// Mitsubishi GX Works2 project: PLC_Group15   PLC: FX3G

// global labels: Global1
VAR_GLOBAL
  StartworkingDay AT X010 : BOOL;
  insertOrange AT D8280 : REAL;
END_VAR
VAR_GLOBAL CONSTANT
  Muiltipy1 : WORD := 100;
  multiply1 : INT;
  divideBy2 : REAL := 2.0;
END_VAR
VAR_GLOBAL
  light AT Y010 : BOOL;
  SampleClemetine AT M2 : BOOL;
  sampleClementine AT D8281 : REAL;
END_VAR
VAR_GLOBAL CONSTANT
  multiply2 : REAL := 100.0;
END_VAR
VAR_GLOBAL
  clemetineInStoreAfterMultiply AT D4005 : REAL;
  checkProportion AT Y006 : BOOL;
  SamplePummels AT X004 : BOOL;
END_VAR
VAR_GLOBAL CONSTANT
  multiply3 : REAL := 100.0;
END_VAR
VAR_GLOBAL
  checkProportion2 AT M42 : BOOL;
  insertClementine AT D8281 : REAL;
  insertPummels AT D8281 : REAL;
  holding AT Y006 : BOOL;
  holding2 AT Y011 : BOOL;
  workingDayLight AT Y010 : BOOL;
  collectFruits AT X002 : BOOL;
END_VAR
VAR_GLOBAL CONSTANT
  washingTimer : REAL := 300.0;
END_VAR
VAR_GLOBAL
  lightOfWashing AT Y005 : BOOL;
  StartingWash AT M7 : BOOL;
END_VAR
VAR_GLOBAL CONSTANT
  const100 : REAL := 100.0;
END_VAR
VAR_GLOBAL
  BiggerThan100 AT M0 : BOOL;
  TakeOnly100 AT M0 : BOOL;
END_VAR
VAR_GLOBAL CONSTANT
  Take100 : REAL := 100.0;
  Take50 : REAL := 50.0;
END_VAR
VAR_GLOBAL
  TurningOnWash AT X002 : BOOL;
  SampleOrange AT M1 : BOOL;
  OrangeSample AT M1 : BOOL;
  ClementineSample AT M2 : BOOL;
  PummelSample AT M3 : BOOL;
  TurnigWashOn AT M4 : BOOL;
  Check100Oranges AT M5 : BOOL;
  Move100 AT M6 : BOOL;
  StartingWash2 AT M7 : BOOL;
  TurningLightWashOn AT M4 : BOOL;
  LessThan100 AT M0 : BOOL;
  MoveLessThan100 AT M8 : BOOL;
END_VAR
VAR_GLOBAL CONSTANT
  Add_150_to_washing_container : INT := 150;
END_VAR
VAR_GLOBAL
  MoveFromStorageToWashing AT X002 : BOOL;
  MoveFromWashingToPress AT X001 : BOOL;
  Collect_Fruits AT X001 : BOOL;
  Keep_Y1_ON AT M18 : BOOL;
  LightForCollecting AT Y001 : BOOL;
END_VAR
VAR_GLOBAL CONSTANT
  Add_100_Oranges : REAL := 100.0;
  Add_50_Clementines : REAL := 50.0;
  Add_50_Pummels : REAL := 50.0;
END_VAR
VAR_GLOBAL
  MoveFruitsToPressContainer AT M9 : BOOL;
  StartPressingProcess AT X011 : BOOL;
  CountingClicks AT CC1 : BOOL;
END_VAR
VAR_GLOBAL CONSTANT
  NumberOfClicks : REAL := 2.0;
END_VAR
VAR_GLOBAL
  Turn_Of_Y1 AT M18 : BOOL;
  StartQA AT X003 : BOOL;
  Sample_AnalogInput2 AT M10 : BOOL;
  CheckValueRange AT M11 : BOOL;
END_VAR
VAR_GLOBAL CONSTANT
  LowerBound : INT := 1;
END_VAR
VAR_GLOBAL
  GE_Than1 AT M12 : BOOL;
  CheckValueRange1 AT M11 : BOOL;
  CheckValueRange2 AT M13 : BOOL;
END_VAR
VAR_GLOBAL CONSTANT
  UpperBound : INT := 5;
  Const1 : REAL := 1.0;
  Const5 : REAL := 5.0;
END_VAR
VAR_GLOBAL
  LE_Than5 AT M14 : BOOL;
  If_M12_ON AT M12 : BOOL;
  If_M14_ON AT M14 : BOOL;
  Timer_Y4_Light AT TC1 : BOOL;
END_VAR
VAR_GLOBAL CONSTANT
  TimerValue : REAL := 500.0;
END_VAR
VAR_GLOBAL
  QA_Light AT Y004 : BOOL;
  Move_Juice_To_Storage AT M15 : BOOL;
  Greater_Than5 AT M12 : BOOL;
  Lower_Than1 AT M14 : BOOL;
  Didnt_Pass_QA AT M16 : BOOL;
  Pass_QA AT M16 : BOOL;
  SampleAgain AT M17 : BOOL;
  Shutting_Y1_Off AT M18 : BOOL;
  FlashingLightsOn AT M18 : BOOL;
  Y2Flash AT Y002 : BOOL;
  Y2Counter AT TC2 : BOOL;
  Turn_Off_Y2 AT TS2 : BOOL;
END_VAR
VAR_GLOBAL CONSTANT
  Const300 : INT := 300;
END_VAR
VAR_GLOBAL
  TurningLightsOn AT M19 : BOOL;
  Y3Counter AT TC3 : BOOL;
  Turn_Off_Y3 AT TS3 : BOOL;
  TurningLightsOff AT TS3 : BOOL;
  CheckValueRange3 AT M20 : BOOL;
  CheckValueRange4 AT M21 : BOOL;
  Greater_Than5_2 AT M22 : BOOL;
  Y3FlashON AT Y003 : BOOL;
  Lower_Than1_22 AT M23 : BOOL;
END_VAR
VAR_GLOBAL CONSTANT
  Const0 : REAL;
END_VAR
VAR_GLOBAL
  NoOrangesInStore AT M24 : BOOL;
  Loop AT M25 : BOOL;
  CheckIfOrange0 AT M26 : BOOL;
  TruncateWashingContainers AT M27 : BOOL;
  TruncateAllFruitStores AT M28 : BOOL;
  Truncate_All_Fruit_Stores AT M28 : BOOL;
  NoOrangesLeft AT M24 : BOOL;
  emergencyExit AT X007 : BOOL;
  X7_Light AT M29 : BOOL;
  MoveToJuiceContainer AT M30 : BOOL;
  EmptyJuice AT M31 : BOOL;
  StartTimerForStorage AT M32 : BOOL;
  CheckJuice AT M33 : BOOL;
  QA1 AT M34 : BOOL;
  Truncate_Juice_Container AT M35 : BOOL;
  insertOranges AT D3000 : REAL;
  OrangesInStore AT D3002 : REAL;
  halfOrange AT D1106 : REAL;
  insertPummel AT D5000 : REAL;
  insertClementines AT D4000 : REAL;
  ClemetinesWashingContainer AT D6002 : REAL;
  PummelsWashingContainer AT D6004 : REAL;
  OrangesWashingContainer AT D6000 : REAL;
  PressContainer AT D6010 : REAL;
  JuiceContainer AT D6012 : REAL;
  SampleAnalogInput2 AT D8281 : INT;
  SaveAnalogOutput AT D6014 : REAL;
  AnalogOutput AT D8282 : INT;
  OrangesAndClementines AT D6008 : REAL;
  StorageContainer AT D6016 : REAL;
  ClementinesInStore AT D4050 : REAL;
  pummelInStore AT D5050 : REAL;
END_VAR
VAR_GLOBAL CONSTANT
  Const2 : INT := 2;
END_VAR
VAR_GLOBAL
  countingWash AT TC0 : BOOL;
END_VAR
VAR_GLOBAL CONSTANT
  Const500 : INT := 500;
END_VAR
VAR_GLOBAL
  Y10_light AT TC4 : BOOL;
  end_day_light AT Y010 : BOOL;
END_VAR
VAR_GLOBAL CONSTANT
  Const_half : INT := 5;
END_VAR
VAR_GLOBAL
  M19Counter AT TC5 : BOOL;
  MoveToJuicer AT TS5 : BOOL;
  SecondQA AT M36 : BOOL;
  Didnt_Pass_QA2 AT M37 : BOOL;
  PassQA_Light AT M38 : BOOL;
  Turn_Lights_Off AT M39 : BOOL;
  Start_QA_Stage AT M40 : BOOL;
  checkProportion1 AT M41 : BOOL;
  checkProportionClementine AT M41 : BOOL;
  checkProportion_2 AT M42 : BOOL;
  Initialize_Y1 AT M43 : BOOL;
  Day_Started AT M44 : BOOL;
  Day_Ended AT M45 : BOOL;
  Initialize_Y10 AT M43 : BOOL;
  Check AT M50 : BOOL;
  MoveToPress AT M45 : BOOL;
  checkTiming AT M51 : BOOL;
  CountingClicksForX11 AT CS1 : BOOL;
  SecondQA_Counter AT CC2 : BOOL;
  CountingWash2 AT TS0 : BOOL;
  SecondQACounter AT CS2 : BOOL;
END_VAR
VAR_GLOBAL CONSTANT
  Const404 : REAL := 404.5;
  Const30 : INT := 30;
  Const10000 : REAL := 10000.0;
END_VAR
VAR_GLOBAL
  Y4Light AT TS1 : BOOL;
END_VAR
VAR_GLOBAL CONSTANT
  Const50 : INT := 50;
END_VAR
VAR_GLOBAL
  Mid_juice_truncate AT M52 : BOOL;
  Close_Y10 AT TS4 : BOOL;
  ClosingTime AT M55 : BOOL;
  FinishCheck1 AT M55 : BOOL;
  FinishCheck2 AT M56 : BOOL;
  MoveAndEmptyPress AT M57 : BOOL;
  FinishedSecondQA AT M58 : BOOL;
  FirstQADone AT M59 : BOOL;
  FirstQA2Done AT M60 : BOOL;
  SecondQADone AT M60 : BOOL;
  SecondQA2Done AT M61 : BOOL;
  tc9 AT TC9 : BOOL;
  ts9 AT TS9 : BOOL;
  Lamp6 AT Y006 : BOOL;
END_VAR
VAR_GLOBAL CONSTANT
  Const_6 : REAL := 6;
  Const_6_int : INT := 6;
  Const_100 : REAL := 100;
END_VAR
VAR_GLOBAL
  FillJuice AT X000 : BOOL;
  StartFillJuice AT M62 : BOOL;
END_VAR
VAR_GLOBAL CONSTANT
  Const_1_5 : REAL := 1.5;
END_VAR
VAR_GLOBAL
  TotalBottles AT D1108 : REAL;
  TimeToFillBottles AT D1110 : INT;
END_VAR
VAR_GLOBAL CONSTANT
  Const_10_int : INT := 10;
  Const_10 : REAL := 10;
END_VAR
VAR_GLOBAL
  checkLessThan10 AT M63 : BOOL;
  LessThan10 AT M64 : BOOL;
  StartLightFillBottles AT M65 : BOOL;
END_VAR
VAR_GLOBAL CONSTANT
  blinkTime : INT := 5;
END_VAR
VAR_GLOBAL
  resetBlink AT M66 : BOOL;
  blink1 AT M67 : BOOL;
  blink2 AT M68 : BOOL;
  tc6 AT TC6 : BOOL;
  ts6 AT TS6 : BOOL;
  tc7 AT TC7 : BOOL;
  ts7 AT TS7 : BOOL;
  tc8 AT TC8 : BOOL;
  ts8 AT TS8 : BOOL;
  Start2blinks AT M69 : BOOL;
  EQto0 AT M70 : BOOL;
END_VAR
VAR_GLOBAL CONSTANT
  Const400 : REAL := 400;
END_VAR

// task Task_01 (event TRUE, interval 0, priority 31): POU_01

PROGRAM POU_01
(* structured ladder/FBD written out as ST: instructions are called as NAME(EN, inputs, outputs); _pN, _eN, _tN stand for wires *)
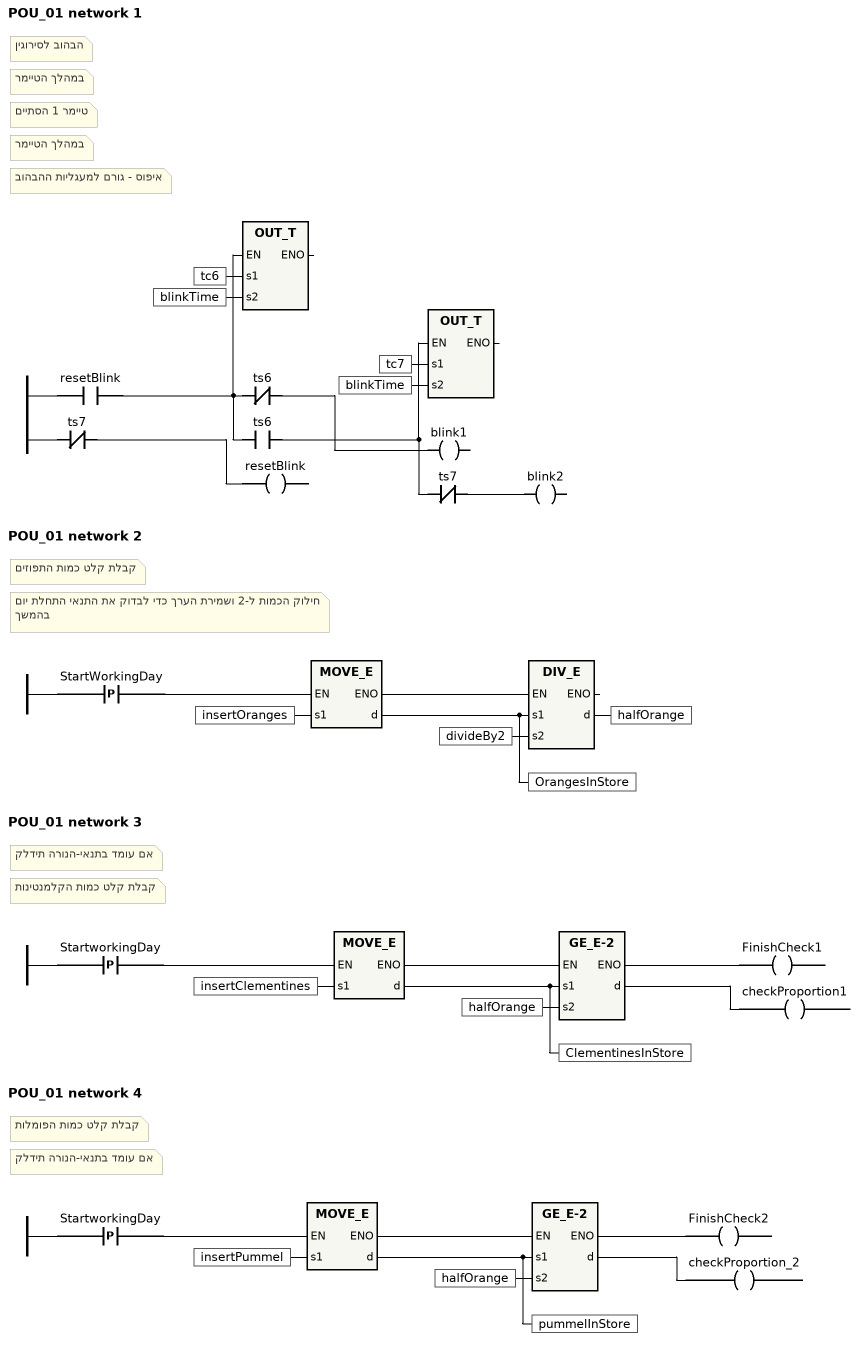
(* network 1 *)
(* הבהוב לסירוגין *)
(* במהלך הטיימר *)
(* טיימר 1 הסתיים *)
(* במהלך הטיימר *)
(* איפוס - גורם למעגליות ההבהוב *)
OUT_T(resetBlink, tc6, blinkTime);
blink1 := resetBlink AND NOT ts6;
_p1 := resetBlink AND ts6;
OUT_T(_p1, tc7, blinkTime);
blink2 := _p1 AND NOT ts7;
resetBlink := NOT ts7;
(* network 2 *)
(* קבלת קלט כמות התפוזים *)
(* חילוק הכמות ל-2 ושמירת הערך כדי לבדוק את התנאי התחלת יום בהמשך *)
_e1 := MOVE_E(LDP(TRUE, StartWorkingDay), insertOranges, OrangesInStore);
DIV_E(_e1, OrangesInStore, divideBy2, halfOrange);
(* network 3 *)
(* אם עומד בתנאי-הנורה תידלק *)
(* קבלת קלט כמות הקלמנטינות *)
_e1 := MOVE_E(LDP(TRUE, StartworkingDay), insertClementines, ClementinesInStore);
_e3 := GE_E(_e1, ClementinesInStore, halfOrange, _t2);
FinishCheck1 := _e3;
checkProportion1 := _t2;
(* network 4 *)
(* קבלת קלט כמות הפומלות *)
(* אם עומד בתנאי-הנורה תידלק *)
_e1 := MOVE_E(LDP(TRUE, StartworkingDay), insertPummel, pummelInStore);
_e3 := GE_E(_e1, pummelInStore, halfOrange, _t2);
FinishCheck2 := _e3;
checkProportion_2 := _t2;
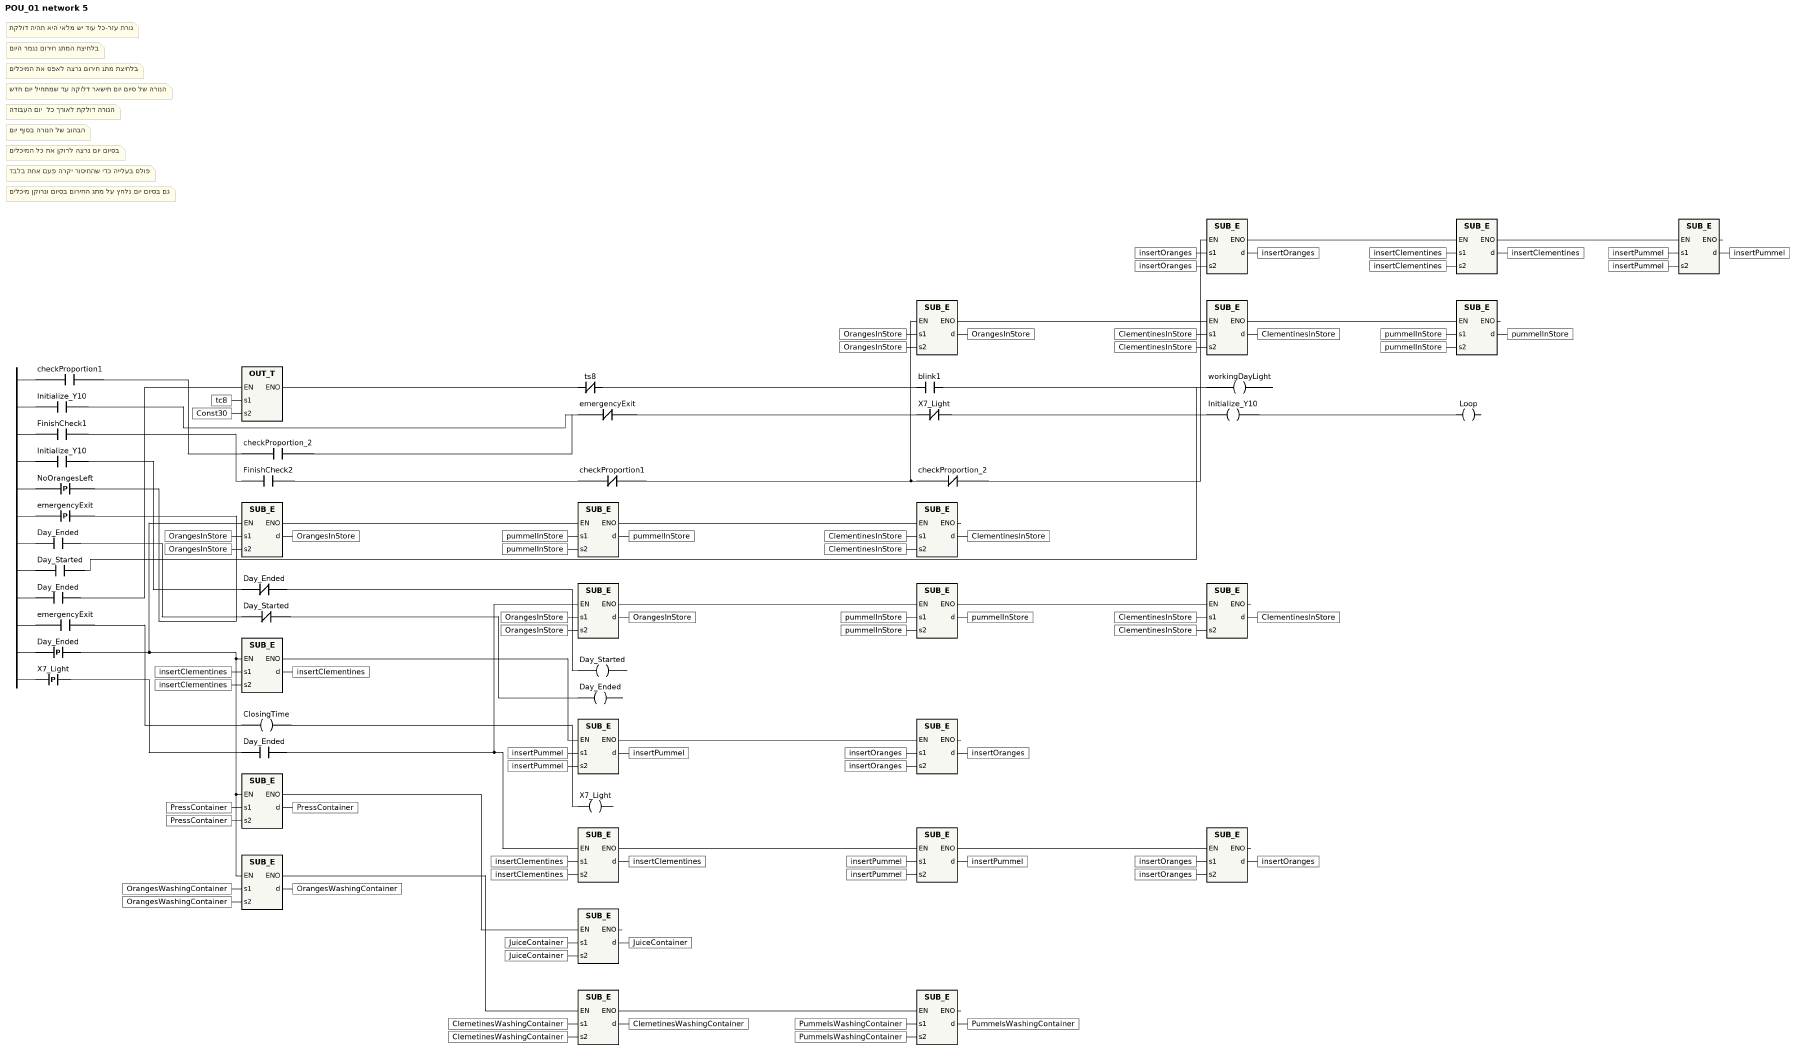
(* network 5 *)
(* נורת עזר-כל עוד יש מלאי היא תהיה דולקת *)
(* בלחיצת המתג חירום נגמר היום *)
(* בלחיצת מתג חירום נרצה לאפס את המיכלים *)
(* הנורה של סיום יום תישאר דלוקה עד שמתחיל יום חדש *)
(* הנורה דולקת לאורך כל  יום העבודה *)
(* הבהוב של הנורה בסוף יום *)
(* בסיום יום נרצה לרוקן את כל המיכלים *)
(* פולס בעלייה כדי שהחיסור יקרה פעם אחת בלבד *)
(* גם בסיום יום נלחץ על מתג החירום בסיום ונרוקן מיכלים *)
_p1 := (((checkProportion1 AND checkProportion_2) OR Initialize_Y10) AND NOT emergencyExit) AND NOT X7_Light;
Initialize_Y10 := _p1;
Loop := _p1;
_p2 := FinishCheck1 AND FinishCheck2 AND NOT checkProportion1;
_e3 := SUB_E(_p2 AND NOT checkProportion_2, insertOranges, insertOranges, insertOranges);
_e4 := SUB_E(_e3, insertClementines, insertClementines, insertClementines);
SUB_E(_e4, insertPummel, insertPummel, insertPummel);
_e5 := SUB_E(_p2, OrangesInStore, OrangesInStore, OrangesInStore);
_e6 := SUB_E(_e5, ClementinesInStore, ClementinesInStore, ClementinesInStore);
SUB_E(_e6, pummelInStore, pummelInStore, pummelInStore);
Day_Started := Initialize_Y10 AND NOT Day_Ended;
Day_Ended := (LDP(TRUE, NoOrangesLeft) OR LDP(TRUE, emergencyExit) OR Day_Ended) AND NOT Day_Started;
_e7 := OUT_T(Day_Ended, tc8, Const30);
workingDayLight := Day_Started OR (_e7 AND NOT ts8 AND blink1);
ClosingTime := emergencyExit;
X7_Light := emergencyExit;
_p8 := LDP(TRUE, Day_Ended);
_e9 := SUB_E(_p8, OrangesInStore, OrangesInStore, OrangesInStore);
_e10 := SUB_E(_e9, pummelInStore, pummelInStore, pummelInStore);
SUB_E(_e10, ClementinesInStore, ClementinesInStore, ClementinesInStore);
_e11 := SUB_E(_p8, insertClementines, insertClementines, insertClementines);
_e12 := SUB_E(_e11, insertPummel, insertPummel, insertPummel);
SUB_E(_e12, insertOranges, insertOranges, insertOranges);
_e13 := SUB_E(_p8, OrangesWashingContainer, OrangesWashingContainer, OrangesWashingContainer);
_e14 := SUB_E(_e13, ClemetinesWashingContainer, ClemetinesWashingContainer, ClemetinesWashingContainer);
SUB_E(_e14, PummelsWashingContainer, PummelsWashingContainer, PummelsWashingContainer);
_e15 := SUB_E(_p8, PressContainer, PressContainer, PressContainer);
SUB_E(_e15, JuiceContainer, JuiceContainer, JuiceContainer);
_p16 := LDP(TRUE, X7_Light) AND Day_Ended;
_e17 := SUB_E(_p16, OrangesInStore, OrangesInStore, OrangesInStore);
_e18 := SUB_E(_e17, pummelInStore, pummelInStore, pummelInStore);
SUB_E(_e18, ClementinesInStore, ClementinesInStore, ClementinesInStore);
_e19 := SUB_E(_p16, insertClementines, insertClementines, insertClementines);
_e20 := SUB_E(_e19, insertPummel, insertPummel, insertPummel);
SUB_E(_e20, insertOranges, insertOranges, insertOranges);
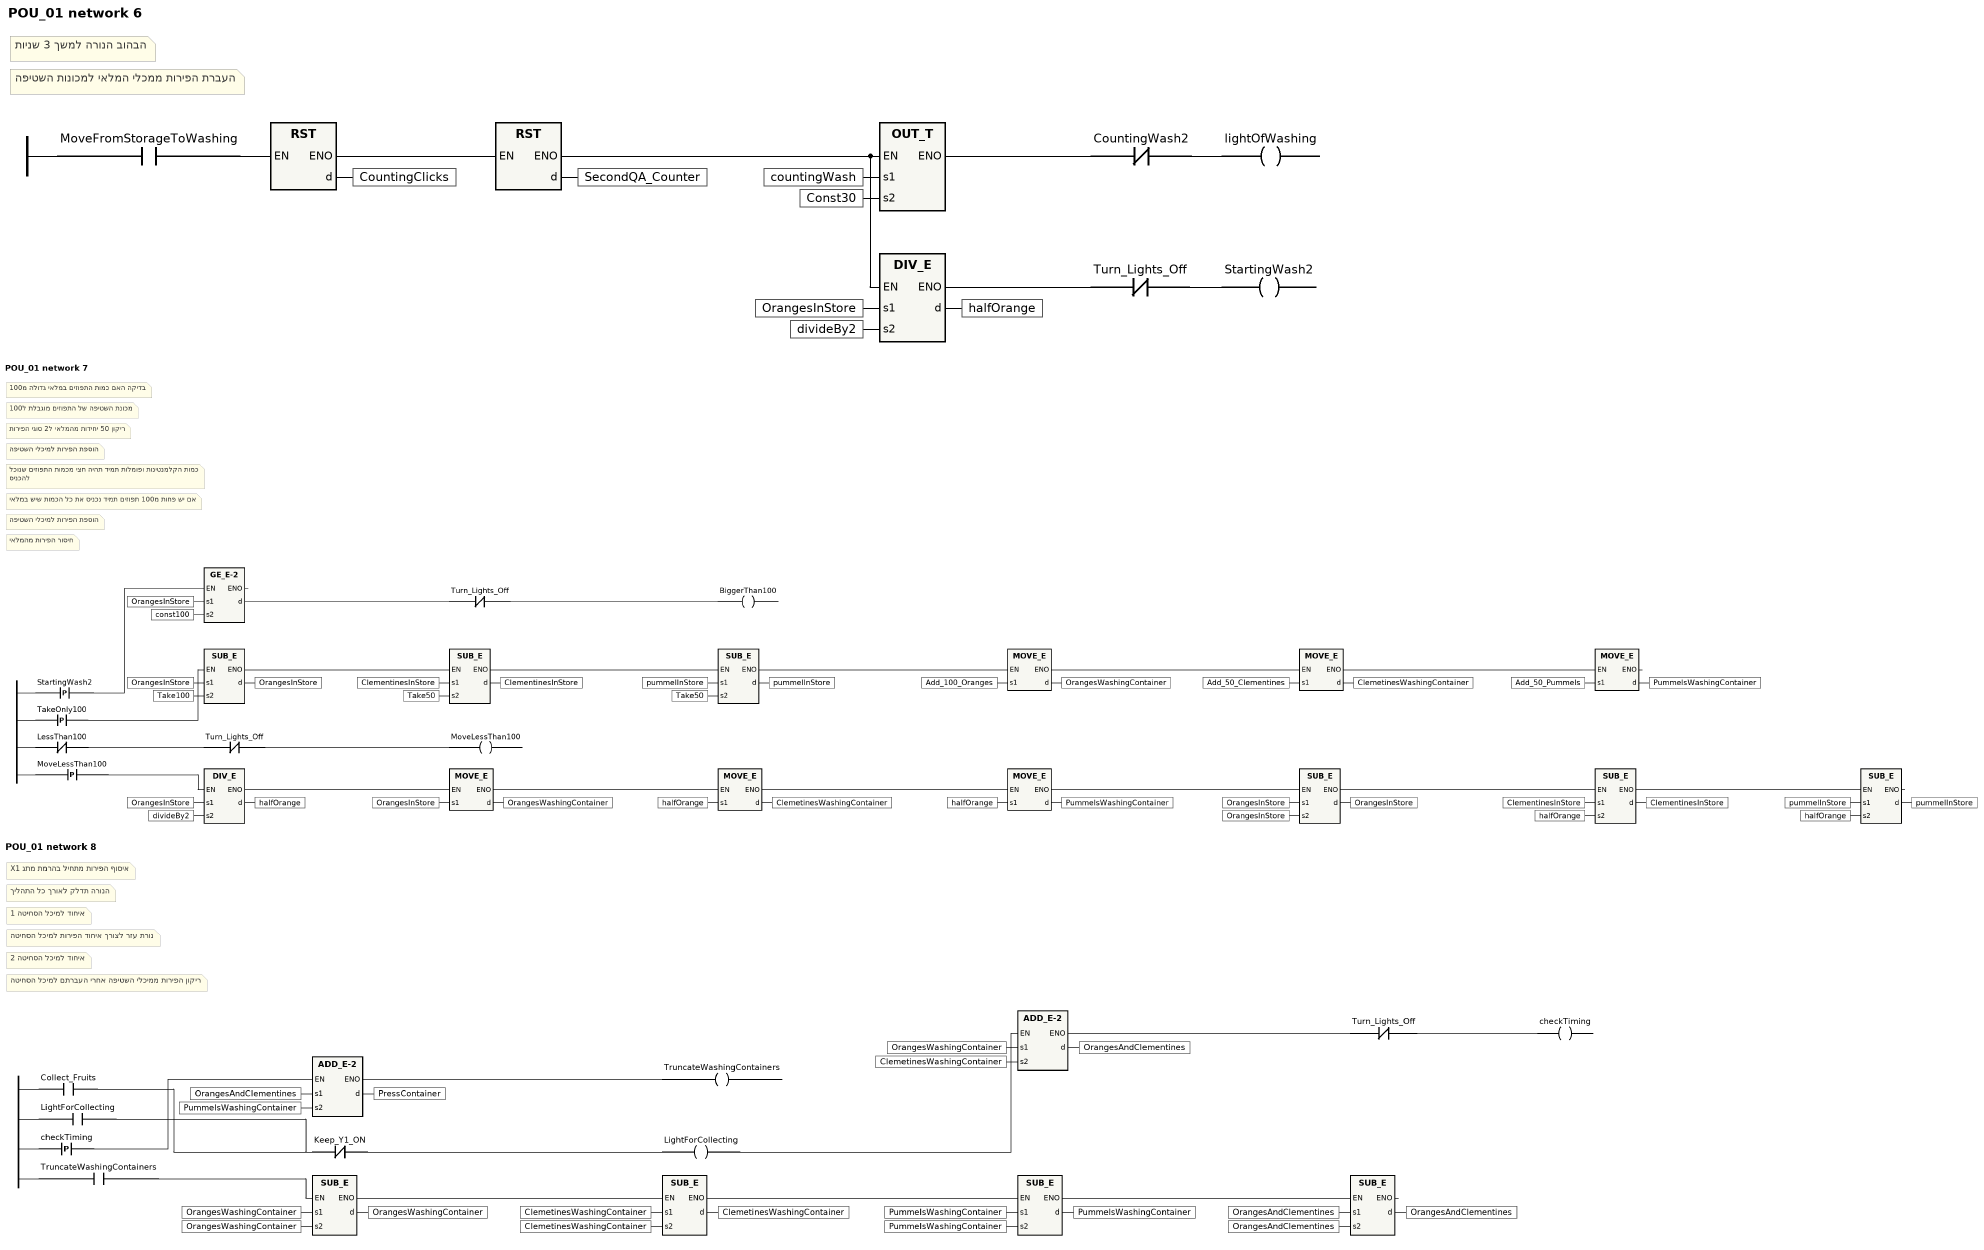
(* network 6 *)
(* הבהוב הנורה למשך 3 שניות *)
(* העברת הפירות ממכלי המלאי למכונות השטיפה *)
_e1 := RST(MoveFromStorageToWashing, CountingClicks);
_e2 := RST(_e1, SecondQA_Counter);
_e3 := OUT_T(_e2, countingWash, Const30);
lightOfWashing := _e3 AND NOT CountingWash2;
_e4 := DIV_E(_e2, OrangesInStore, divideBy2, halfOrange);
StartingWash2 := _e4 AND NOT Turn_Lights_Off;
(* network 7 *)
(* בדיקה האם כמות התפוזים במלאי גדולה מ100 *)
(* מכונת השטיפה של התפוזים מוגבלת ל100 *)
(* ריקון 50 יחידות מהמלאי ל2 סוגי הפירות *)
(* הוספת הפירות למיכלי השטיפה *)
(* כמות הקלמנטינות ופומלות תמיד תהיה חצי מכמות התפוזים שנוכל להכניס *)
(* אם יש פחות מ100 תפוזים תמיד נכניס את כל הכמות שיש במלאי *)
(* הוספת הפירות למיכלי השטיפה *)
(* חיסור הפירות מהמלאי *)
GE_E(LDP(TRUE, StartingWash2), OrangesInStore, const100, _t1);
BiggerThan100 := _t1 AND NOT Turn_Lights_Off;
_e2 := SUB_E(LDP(TRUE, TakeOnly100), OrangesInStore, Take100, OrangesInStore);
_e3 := SUB_E(_e2, ClementinesInStore, Take50, ClementinesInStore);
_e4 := SUB_E(_e3, pummelInStore, Take50, pummelInStore);
_e5 := MOVE_E(_e4, Add_100_Oranges, OrangesWashingContainer);
_e6 := MOVE_E(_e5, Add_50_Clementines, ClemetinesWashingContainer);
MOVE_E(_e6, Add_50_Pummels, PummelsWashingContainer);
MoveLessThan100 := NOT LessThan100 AND NOT Turn_Lights_Off;
_e7 := DIV_E(LDP(TRUE, MoveLessThan100), OrangesInStore, divideBy2, halfOrange);
_e8 := MOVE_E(_e7, OrangesInStore, OrangesWashingContainer);
_e9 := MOVE_E(_e8, halfOrange, ClemetinesWashingContainer);
_e10 := MOVE_E(_e9, halfOrange, PummelsWashingContainer);
_e11 := SUB_E(_e10, OrangesInStore, OrangesInStore, OrangesInStore);
_e12 := SUB_E(_e11, ClementinesInStore, halfOrange, ClementinesInStore);
SUB_E(_e12, pummelInStore, halfOrange, pummelInStore);
(* network 8 *)
(* איסוף הפירות מתחיל בהרמת מתג X1 *)
(* הנורה תדלק לאורך כל התהליך *)
(* איחוד למיכל הסחיטה 1 *)
(* נורת עזר לצורך איחוד הפירות למיכל הסחיטה *)
(* איחוד למיכל הסחיטה 2 *)
(* ריקון הפירות ממיכלי השטיפה אחרי העברתם למיכל הסחיטה *)
_p1 := (Collect_Fruits OR LightForCollecting) AND NOT Keep_Y1_ON;
LightForCollecting := _p1;
_e2 := ADD_E(_p1, OrangesWashingContainer, ClemetinesWashingContainer, OrangesAndClementines);
checkTiming := _e2 AND NOT Turn_Lights_Off;
_e3 := ADD_E(LDP(TRUE, checkTiming), OrangesAndClementines, PummelsWashingContainer, PressContainer);
TruncateWashingContainers := _e3;
_e4 := SUB_E(TruncateWashingContainers, OrangesWashingContainer, OrangesWashingContainer, OrangesWashingContainer);
_e5 := SUB_E(_e4, ClemetinesWashingContainer, ClemetinesWashingContainer, ClemetinesWashingContainer);
_e6 := SUB_E(_e5, PummelsWashingContainer, PummelsWashingContainer, PummelsWashingContainer);
SUB_E(_e6, OrangesAndClementines, OrangesAndClementines, OrangesAndClementines);
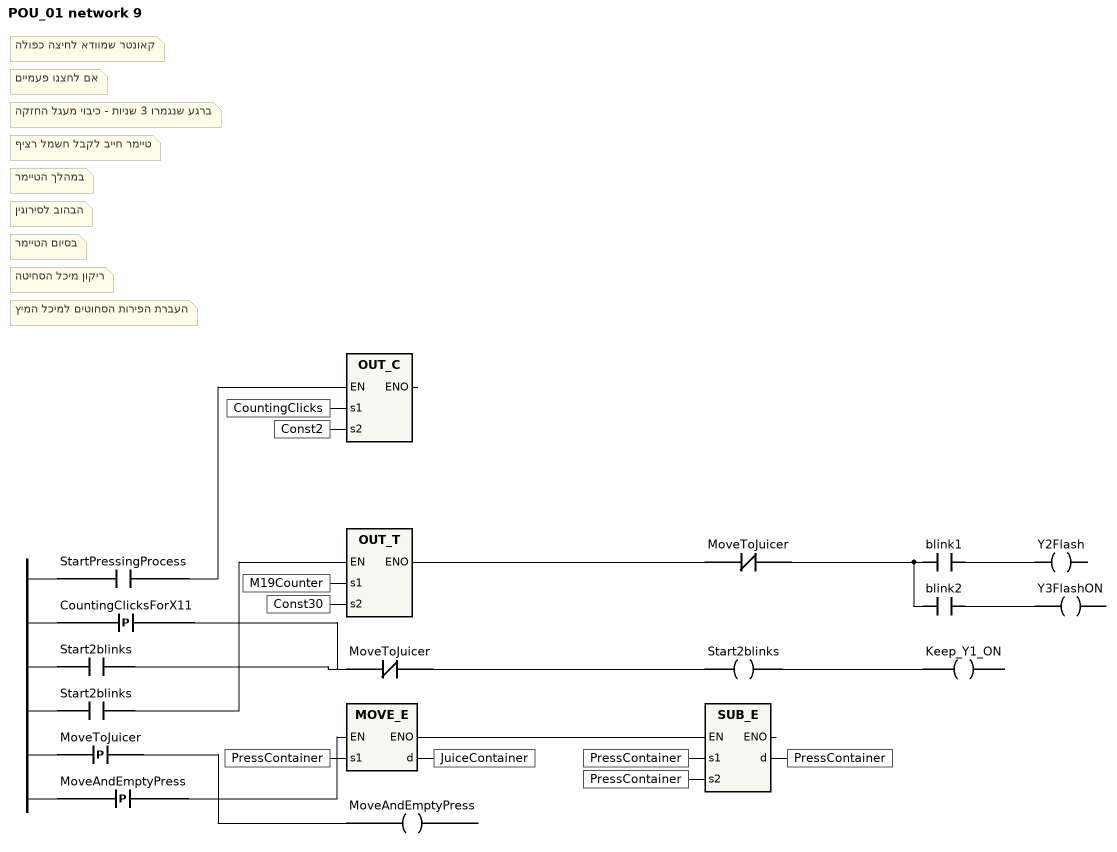
(* network 9 *)
(* קאונטר שמוודא לחיצה כפולה *)
(* אם לחצנו פעמיים *)
(* ברגע שנגמרו 3 שניות - כיבוי מעגל החזקה *)
(* טיימר חייב לקבל חשמל רציף *)
(* במהלך הטיימר *)
(* הבהוב לסירוגין *)
(* בסיום הטיימר *)
(* ריקון מיכל הסחיטה *)
(* העברת הפירות הסחוטים למיכל המיץ *)
OUT_C(StartPressingProcess, CountingClicks, Const2);
_p1 := (LDP(TRUE, CountingClicksForX11) OR Start2blinks) AND NOT MoveToJuicer;
Start2blinks := _p1;
Keep_Y1_ON := _p1;
_e2 := OUT_T(Start2blinks, M19Counter, Const30);
_p3 := _e2 AND NOT MoveToJuicer;
Y2Flash := _p3 AND blink1;
Y3FlashON := _p3 AND blink2;
MoveAndEmptyPress := LDP(TRUE, MoveToJuicer);
_e4 := MOVE_E(LDP(TRUE, MoveAndEmptyPress), PressContainer, JuiceContainer);
SUB_E(_e4, PressContainer, PressContainer, PressContainer);
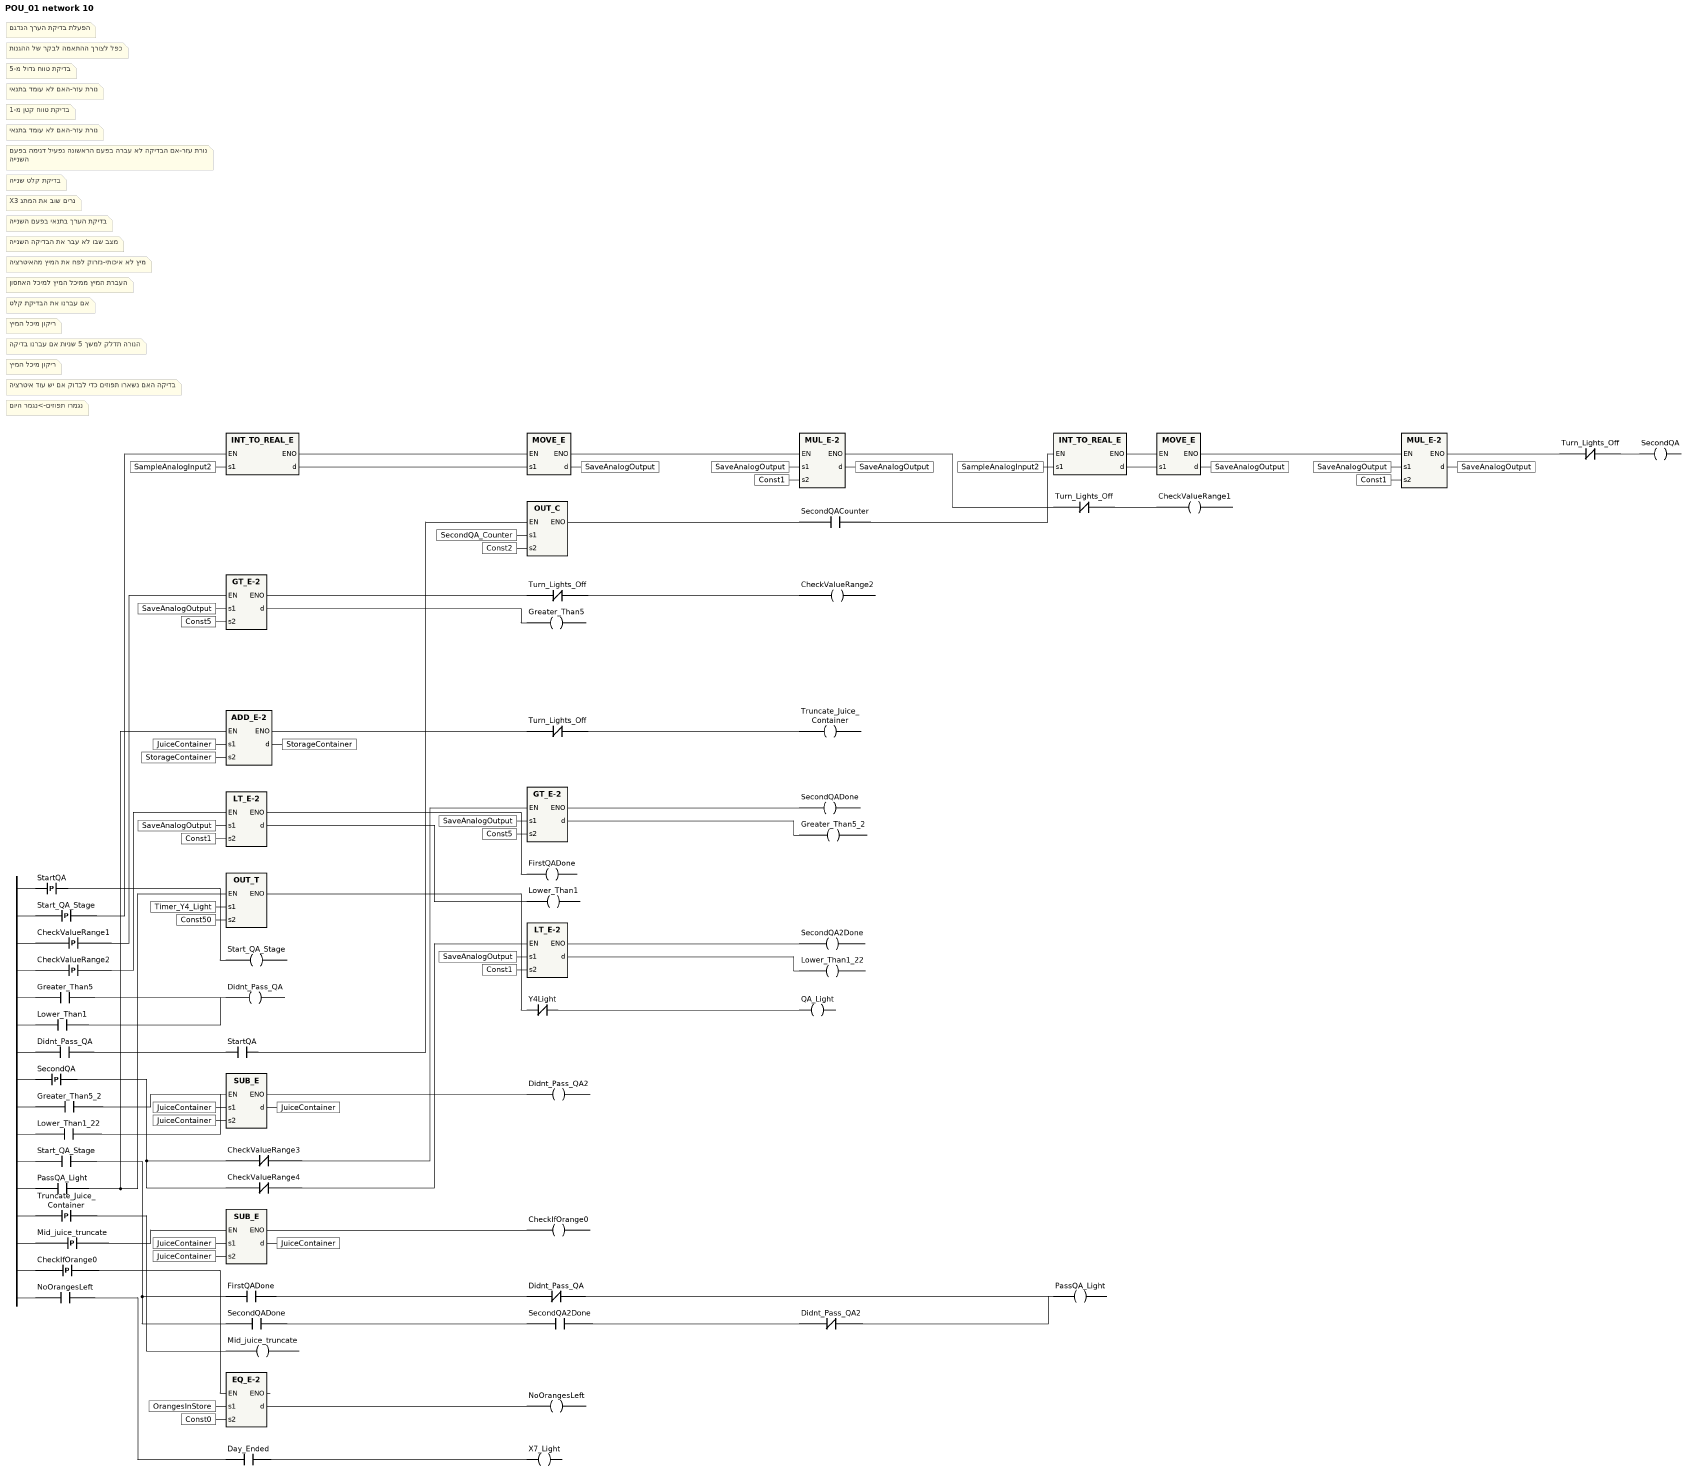
(* network 10 *)
(* הפעלת בדיקת הערך הנדגם *)
(* כפל לצורך ההתאמה לבקר של ההגנות *)
(* בדיקת טווח גדול מ-5 *)
(* נורת עזר-האם לא עומד בתנאי *)
(* בדיקת טווח קטן מ-1 *)
(* נורת עזר-האם לא עומד בתנאי *)
(* נורת עזר-אם הבדיקה לא עברה בפעם הראשונה נפעיל דגימה בפעם השנייה *)
(* בדיקת קלט שנייה *)
(* נרים שוב את המתג X3 *)
(* בדיקת הערך בתנאי בפעם השנייה *)
(* מצב שבו לא עבר את הבדיקה השנייה *)
(* מיץ לא איכותי-נזרוק לפח את המיץ מהאיטרציה *)
(* העברת המיץ ממיכל המיץ למיכל האחסון *)
(* אם עברנו את הבדיקת קלט *)
(* ריקון מיכל המיץ *)
(* הנורה תדלק למשך 5 שניות אם עברנו בדיקה *)
(* ריקון מיכל המיץ *)
(* בדיקה האם נשארו תפוזים כדי לבדוק אם יש עוד איטרציה *)
(* נגמרו תפוזים->נגמר היום *)
Start_QA_Stage := LDP(TRUE, StartQA);
_e2 := INT_TO_REAL_E(LDP(TRUE, Start_QA_Stage), SampleAnalogInput2, _t1);
_e3 := MOVE_E(_e2, _t1, SaveAnalogOutput);
_e4 := MUL_E(_e3, SaveAnalogOutput, Const1, SaveAnalogOutput);
CheckValueRange1 := _e4 AND NOT Turn_Lights_Off;
_e6 := GT_E(LDP(TRUE, CheckValueRange1), SaveAnalogOutput, Const5, _t5);
CheckValueRange2 := _e6 AND NOT Turn_Lights_Off;
Greater_Than5 := _t5;
_e8 := LT_E(LDP(TRUE, CheckValueRange2), SaveAnalogOutput, Const1, _t7);
FirstQADone := _e8;
Lower_Than1 := _t7;
Didnt_Pass_QA := Greater_Than5 OR Lower_Than1;
_e9 := OUT_C(Didnt_Pass_QA AND StartQA, SecondQA_Counter, Const2);
_e11 := INT_TO_REAL_E(_e9 AND SecondQACounter, SampleAnalogInput2, _t10);
_e12 := MOVE_E(_e11, _t10, SaveAnalogOutput);
_e13 := MUL_E(_e12, SaveAnalogOutput, Const1, SaveAnalogOutput);
SecondQA := _e13 AND NOT Turn_Lights_Off;
_p14 := LDP(TRUE, SecondQA);
_e16 := GT_E(_p14 AND NOT CheckValueRange3, SaveAnalogOutput, Const5, _t15);
SecondQADone := _e16;
Greater_Than5_2 := _t15;
_e18 := LT_E(_p14 AND NOT CheckValueRange4, SaveAnalogOutput, Const1, _t17);
SecondQA2Done := _e18;
Lower_Than1_22 := _t17;
_e19 := SUB_E(Greater_Than5_2 OR Lower_Than1_22, JuiceContainer, JuiceContainer, JuiceContainer);
Didnt_Pass_QA2 := _e19;
PassQA_Light := (Start_QA_Stage AND FirstQADone AND NOT Didnt_Pass_QA) OR (Start_QA_Stage AND SecondQADone AND SecondQA2Done AND NOT Didnt_Pass_QA2);
_e20 := ADD_E(PassQA_Light, JuiceContainer, StorageContainer, StorageContainer);
Truncate_Juice_Container := _e20 AND NOT Turn_Lights_Off;
_e21 := OUT_T(PassQA_Light, Timer_Y4_Light, Const50);
QA_Light := _e21 AND NOT Y4Light;
Mid_juice_truncate := LDP(TRUE, Truncate_Juice_Container);
_e22 := SUB_E(LDP(TRUE, Mid_juice_truncate), JuiceContainer, JuiceContainer, JuiceContainer);
CheckIfOrange0 := _e22;
EQ_E(LDP(TRUE, CheckIfOrange0), OrangesInStore, Const0, _t23);
NoOrangesLeft := _t23;
X7_Light := NoOrangesLeft AND Day_Ended;
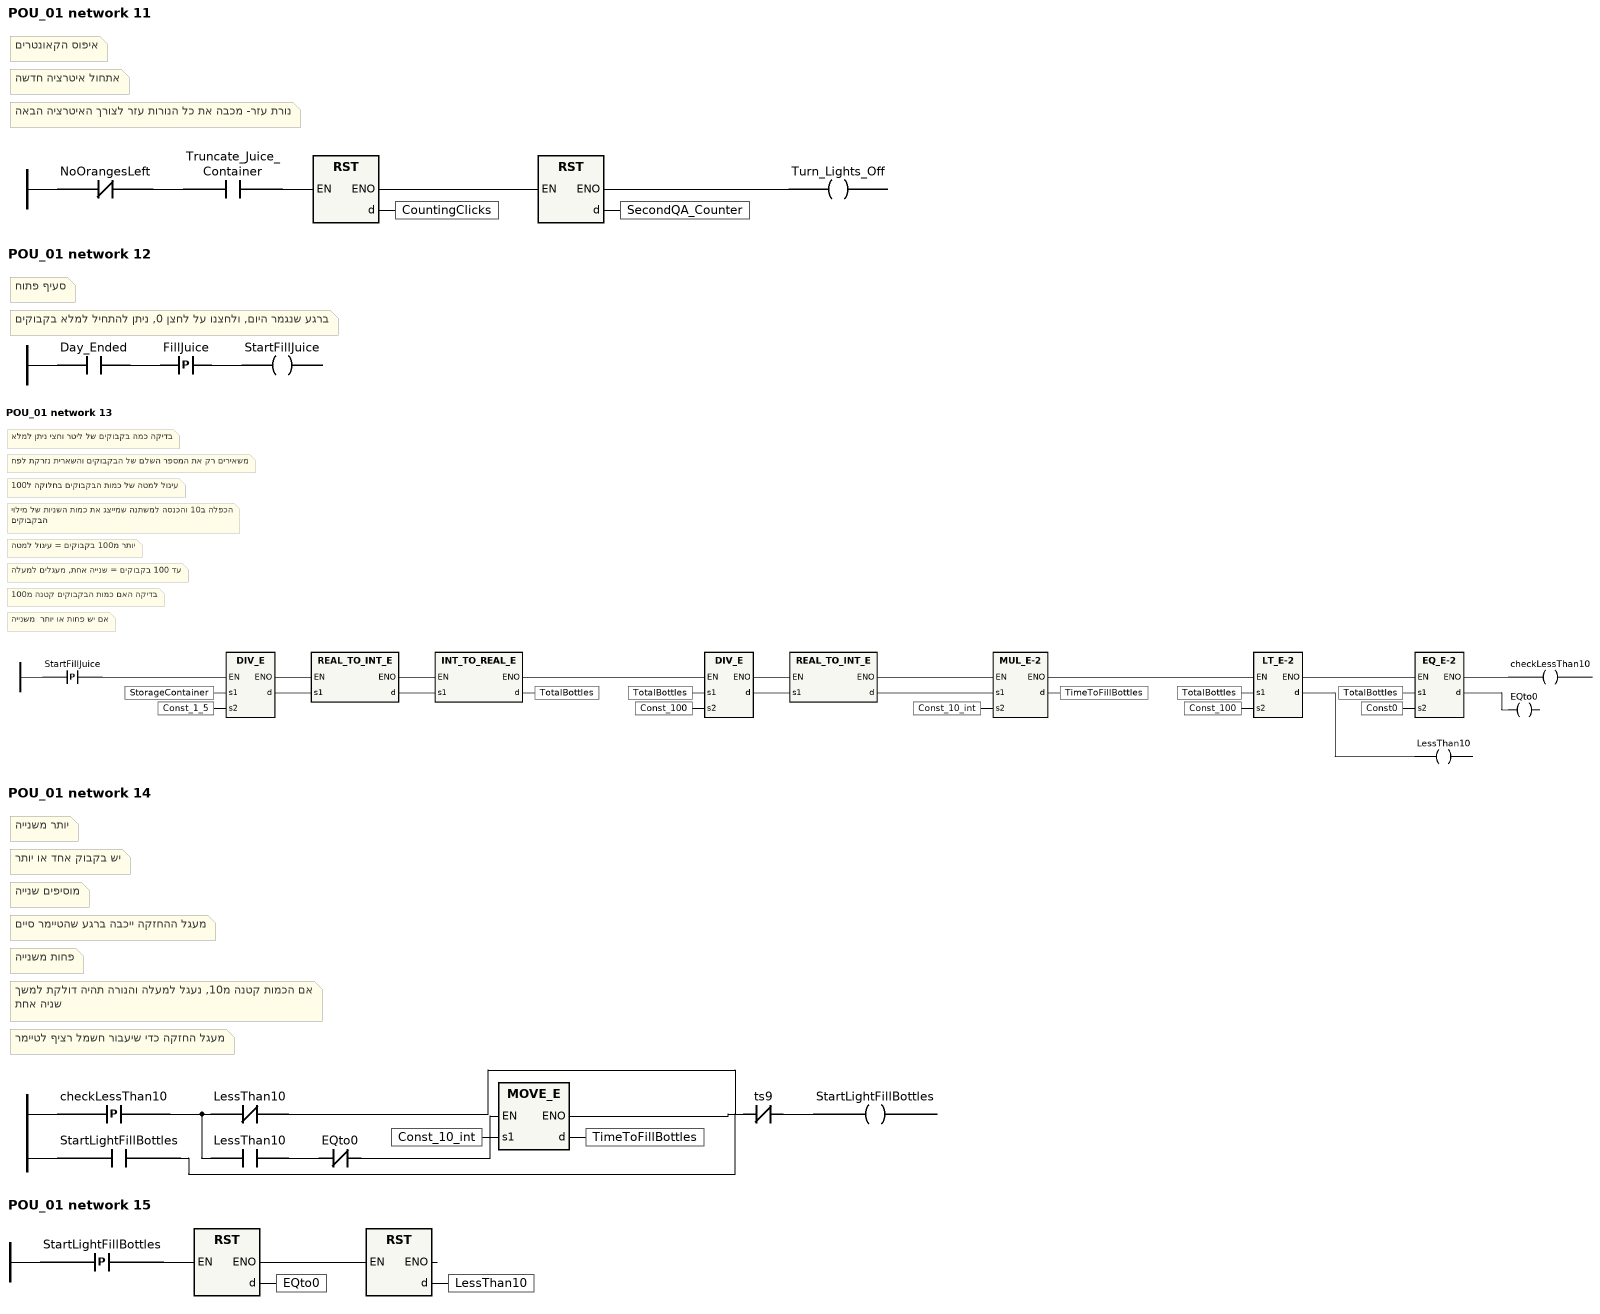
(* network 11 *)
(* איפוס הקאונטרים *)
(* אתחול איטרציה חדשה *)
(* נורת עזר- מכבה את כל הנורות עזר לצורך האיטרציה הבאה *)
_e1 := RST(NOT NoOrangesLeft AND Truncate_Juice_Container, CountingClicks);
_e2 := RST(_e1, SecondQA_Counter);
Turn_Lights_Off := _e2;
(* network 12 *)
(* סעיף פתוח *)
(* ברגע שנגמר היום, ולחצנו על לחצן 0, ניתן להתחיל למלא בקבוקים *)
StartFillJuice := Day_Ended AND LDP(TRUE, FillJuice);
(* network 13 *)
(* בדיקה כמה בקבוקים של ליטר וחצי ניתן למלא *)
(* משאירים רק את המספר השלם של הבקבוקים והשארית נזרקת לפח *)
(* עיגול למטה של כמות הבקבוקים בחלוקה ל100 *)
(* הכפלה ב10 והכנסה למשתנה שמייצג את כמות השניות של מילוי הבקבוקים *)
(* יותר מ100 בקבוקים = עיגול למטה *)
(* עד 100 בקבוקים = שנייה אחת, מעגלים למעלה *)
(* בדיקה האם כמות הבקבוקים קטנה מ100 *)
(* אם יש פחות או יותר  משנייה *)
_e2 := DIV_E(LDP(TRUE, StartFillJuice), StorageContainer, Const_1_5, _t1);
_e4 := REAL_TO_INT_E(_e2, _t1, _t3);
_e5 := INT_TO_REAL_E(_e4, _t3, TotalBottles);
_e7 := DIV_E(_e5, TotalBottles, Const_100, _t6);
_e9 := REAL_TO_INT_E(_e7, _t6, _t8);
_e10 := MUL_E(_e9, _t8, Const_10_int, TimeToFillBottles);
_e12 := LT_E(_e10, TotalBottles, Const_100, _t11);
_e14 := EQ_E(_e12, TotalBottles, Const0, _t13);
checkLessThan10 := _e14;
LessThan10 := _t11;
EQto0 := _t13;
(* network 14 *)
(* יותר משנייה *)
(* יש בקבוק אחד או יותר *)
(* מוסיפים שנייה *)
(* מעגל ההחזקה ייכבה ברגע שהטיימר סיים *)
(* פחות משנייה *)
(* אם הכמות קטנה מ10, נעגל למעלה והנורה תהיה דולקת למשך שניה אחת *)
(* מעגל החזקה כדי שיעבור חשמל רציף לטיימר *)
_p1 := LDP(TRUE, checkLessThan10);
_e2 := MOVE_E(_p1 AND LessThan10 AND NOT EQto0, Const_10_int, TimeToFillBottles);
StartLightFillBottles := ((_p1 AND NOT LessThan10) OR _e2 OR StartLightFillBottles) AND NOT ts9;
(* network 15 *)
_e1 := RST(LDP(TRUE, StartLightFillBottles), EQto0);
RST(_e1, LessThan10);
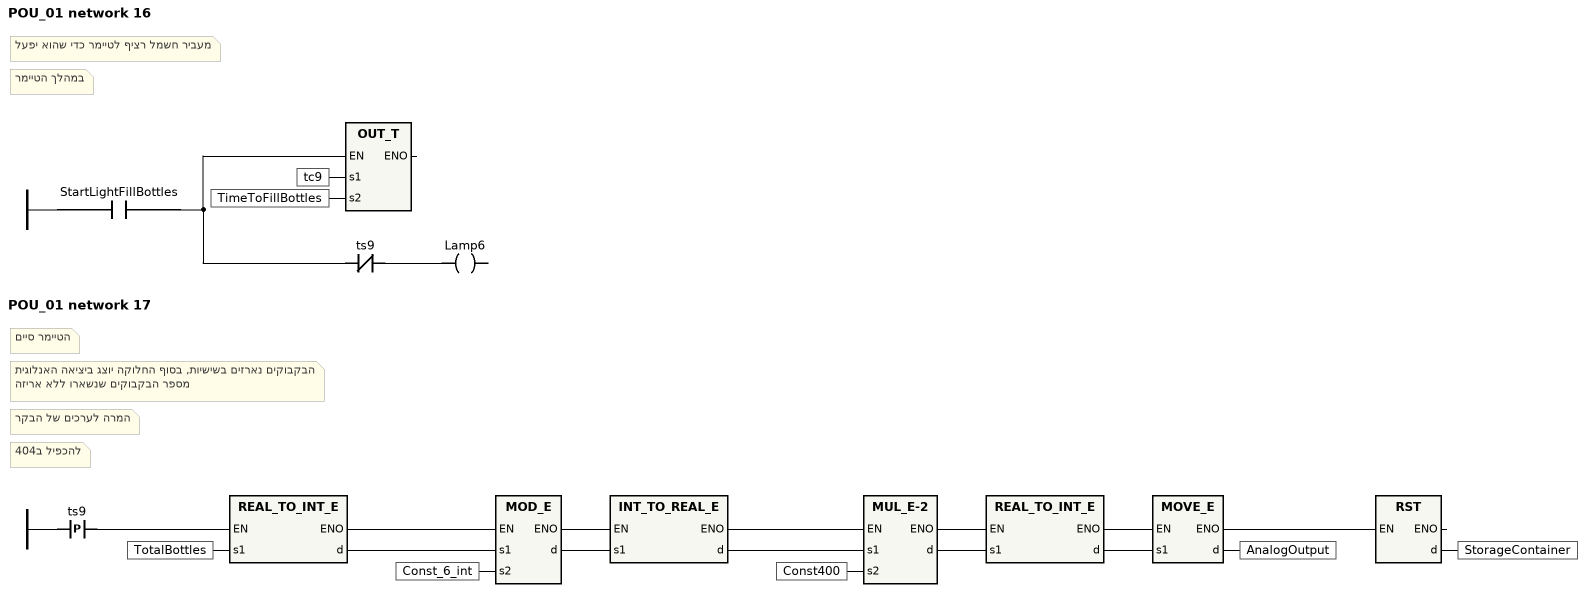
(* network 16 *)
(* מעביר חשמל רציף לטיימר כדי שהוא יפעל *)
(* במהלך הטיימר *)
OUT_T(StartLightFillBottles, tc9, TimeToFillBottles);
Lamp6 := StartLightFillBottles AND NOT ts9;
(* network 17 *)
(* הטיימר סיים *)
(* הבקבוקים נארזים בשישיות, בסוף החלוקה יוצג ביציאה האנלוגית מספר הבקבוקים שנשארו ללא אריזה *)
(* המרה לערכים של הבקר *)
(* להכפיל ב404 *)
_e2 := REAL_TO_INT_E(LDP(TRUE, ts9), TotalBottles, _t1);
_e4 := MOD_E(_e2, _t1, Const_6_int, _t3);
_e6 := INT_TO_REAL_E(_e4, _t3, _t5);
_e8 := MUL_E(_e6, _t5, Const400, _t7);
_e10 := REAL_TO_INT_E(_e8, _t7, _t9);
_e11 := MOVE_E(_e10, _t9, AnalogOutput);
RST(_e11, StorageContainer);
END_PROGRAM
